(* CoDeSys 2.3 export: MANUAL_ALMACEN.EXP *)

(* POU Manual/Manual_Almacen, LD *)
PROGRAM Manual_Almacen
VAR
END_VAR
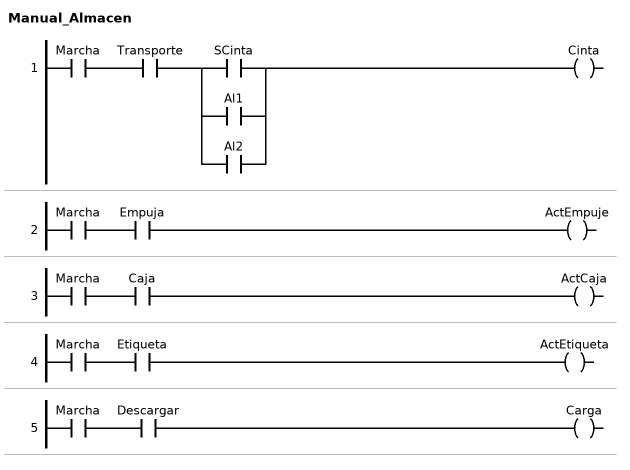
_LD_ (* Ladder Diagram *)
NETWORK 1
	[Marcha] - [Transporte] - { [SCinta] | [Al1] | [Al2] } --- (Cinta)
NETWORK 2
	[Marcha] - [Empuja] --- (ActEmpuje)
NETWORK 3
	[Marcha] - [Caja] --- (ActCaja)
NETWORK 4
	[Marcha] - [Etiqueta] --- (ActEtiqueta)
NETWORK 5
	[Marcha] - [Descargar] --- (Carga)
_END_LD_
(* the same logic as Structured Text *)
(* Network 1 *)
Cinta := Marcha AND Transporte AND (SCinta OR Al1 OR Al2);
(* Network 2 *)
ActEmpuje := Marcha AND Empuja;
(* Network 3 *)
ActCaja := Marcha AND Caja;
(* Network 4 *)
ActEtiqueta := Marcha AND Etiqueta;
(* Network 5 *)
Carga := Marcha AND Descargar;
END_PROGRAM
